(* Schneider Machine Expert - Basic project schnider sensor plc, file version 2.7.0.0 *)
(* ProjectInformations: Name=New project *)

HARDWARE
  Cpu 0: TM200C24R
  EthernetConfiguration: NetworkName=M200, IpAllocationMode=FixedAddress, IpAddress=0.0.0.0, SubnetMask=0.0.0.0
  SerialLineConfiguration: Baud=Baud19200, Parity=ParityEven, DataBits=DataBits8, StopBits=StopBits1, PhysicalMedium=PhysicalMediumRs485, TransmissionMode=TransmissionModeModbusRtu, SlaveId=1, Addressing=SlaveAddressing
  MastTask: UsePeriodScanMode=false, PeriodScan=100
  FastTask: Period=255
  CpuBehavior: StartingMode=StartAsPreviousState, AutoSaveRamOnEeprom=true, WatchdogPeriod=250

SYMBOLS  (address, symbol, comment, settings)
  %M0         "x"
  %M1         "mm1"
  %M2         "msensor"
  %M3         "msensor stop"
  %M4         "mm1"
  %M6         "mtimer"
  %TM0        [Preset=5, Base=OneSecond]
  %I0.0       "start"
  %I0.1       "stop"
  %I0.2       "sensor"
  %Q0.0       "m1"

POU New POU
  (* SectionNumber=1 *)

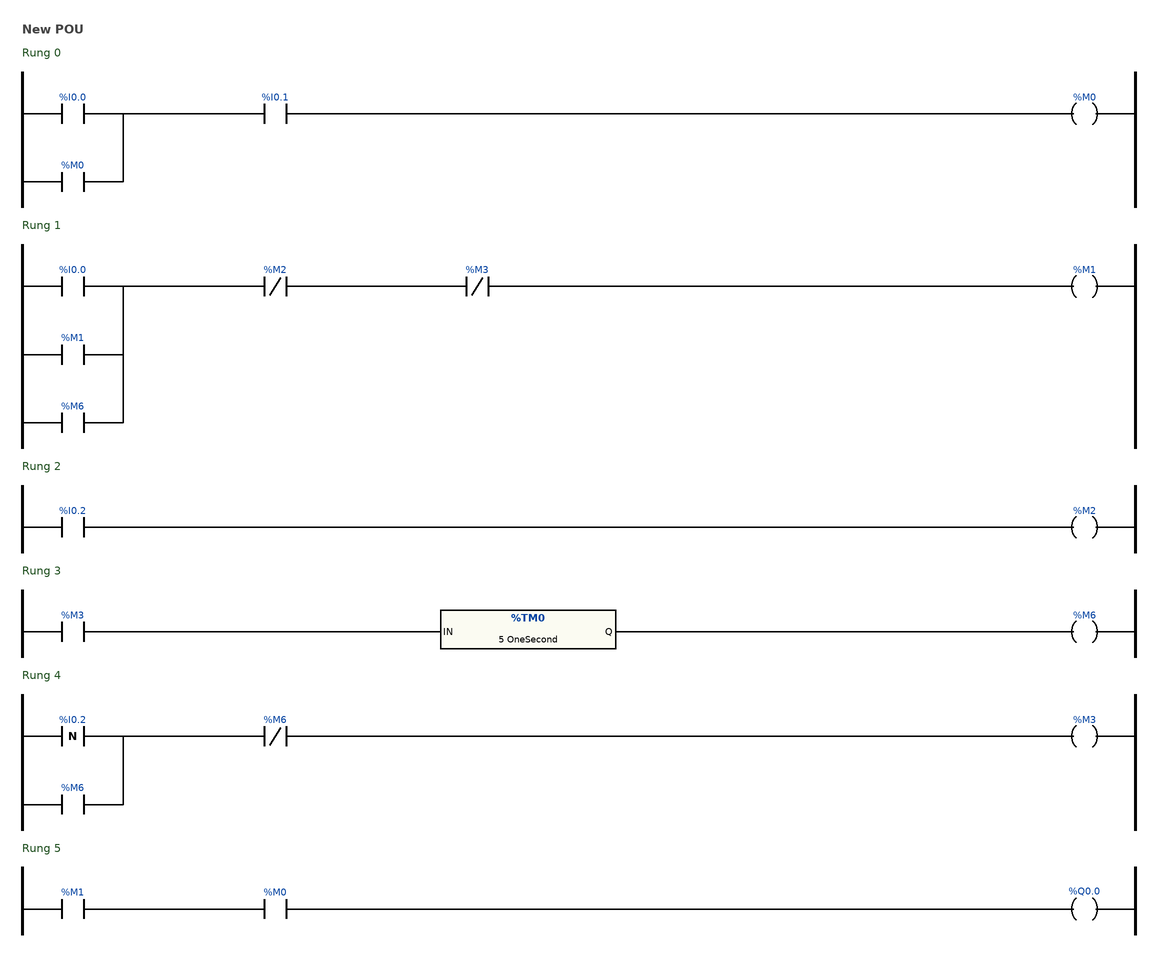

// Rung 0
  LD %I0.0
  OR %M0
  AND %I0.1
  ST %M0
  // as ST:
  //   %M0 := (%I0.0 OR %M0) AND %I0.1;

// Rung 1
  LD %I0.0
  OR %M1
  OR %M6
  ANDN %M2
  ANDN %M3
  ST %M1
  // as ST:
  //   %M1 := (%I0.0 OR %M1 OR %M6) AND NOT %M2 AND NOT %M3;

// Rung 2
  LD %I0.2
  ST %M2
  // as ST:
  //   %M2 := %I0.2;

// Rung 3
  BLK %TM0
  LD %M3
  IN
  OUT_BLK
  LD Q
  ST %M6
  END_BLK
  // as ST:
  //   %TM0(IN := %M3);
  //   %M6 := %TM0.Q;

// Rung 4
  LDF %I0.2
  OR %M6
  ANDN %M6
  ST %M3
  // as ST:
  //   %M3 := (FALLING(%I0.2) OR %M6) AND NOT %M6;

// Rung 5
  LD %M1
  AND %M0
  ST %Q0.0
  // as ST:
  //   %Q0.0 := %M1 AND %M0;
